REGION Network 2: TESTE CHACHA 20 ROUNDS
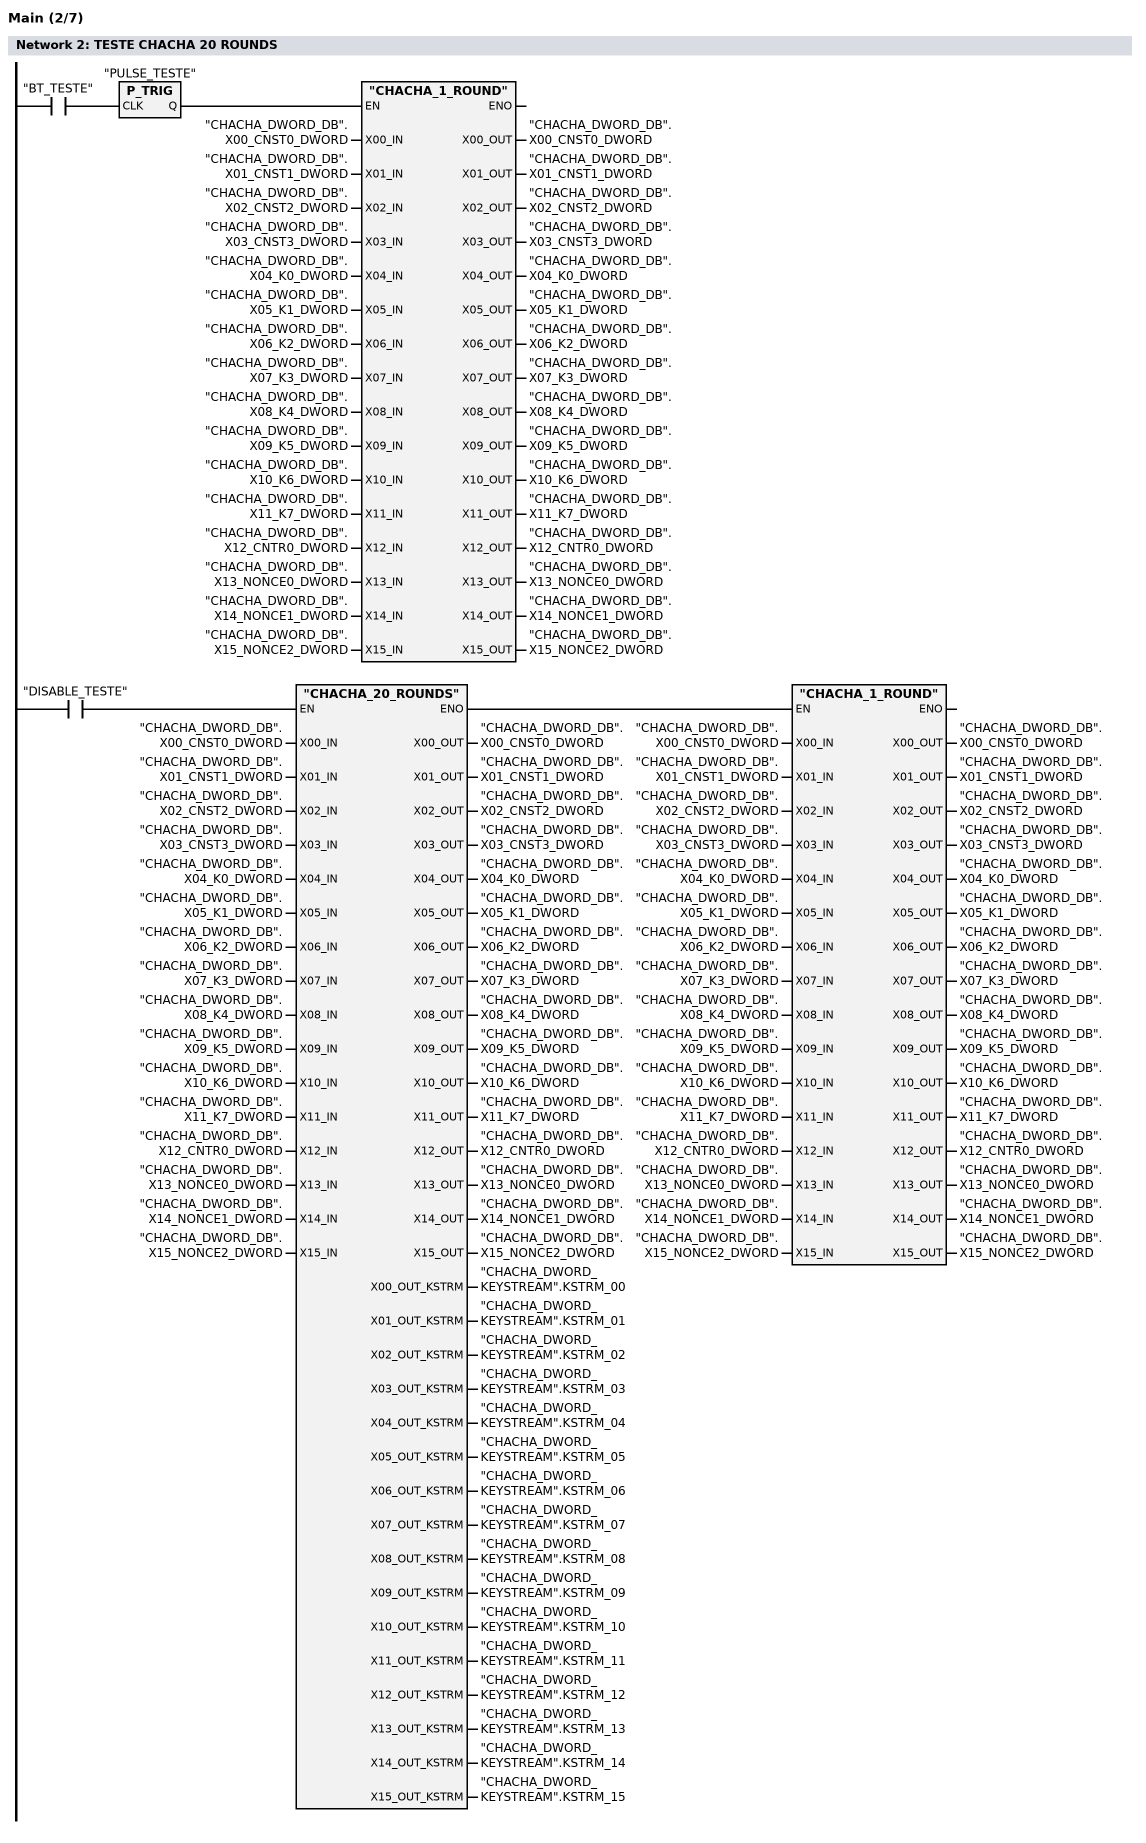
   RUNG wire#powerrail
      Contact( "BT_TESTE" )
      P_Trig( "PULSE_TESTE" )
      "CHACHA_1_ROUND"(X00_IN := "CHACHA_DWORD_DB".X00_CNST0_DWORD, X01_IN := "CHACHA_DWORD_DB".X01_CNST1_DWORD, X02_IN := "CHACHA_DWORD_DB".X02_CNST2_DWORD, X03_IN := "CHACHA_DWORD_DB".X03_CNST3_DWORD, X04_IN := "CHACHA_DWORD_DB".X04_K0_DWORD, X05_IN := "CHACHA_DWORD_DB".X05_K1_DWORD, X06_IN := "CHACHA_DWORD_DB".X06_K2_DWORD, X07_IN := "CHACHA_DWORD_DB".X07_K3_DWORD, X08_IN := "CHACHA_DWORD_DB".X08_K4_DWORD, X09_IN := "CHACHA_DWORD_DB".X09_K5_DWORD, X10_IN := "CHACHA_DWORD_DB".X10_K6_DWORD, X11_IN := "CHACHA_DWORD_DB".X11_K7_DWORD, X12_IN := "CHACHA_DWORD_DB".X12_CNTR0_DWORD, X13_IN := "CHACHA_DWORD_DB".X13_NONCE0_DWORD, X14_IN := "CHACHA_DWORD_DB".X14_NONCE1_DWORD, X15_IN := "CHACHA_DWORD_DB".X15_NONCE2_DWORD, X00_OUT => "CHACHA_DWORD_DB".X00_CNST0_DWORD, X01_OUT => "CHACHA_DWORD_DB".X01_CNST1_DWORD, X02_OUT => "CHACHA_DWORD_DB".X02_CNST2_DWORD, X03_OUT => "CHACHA_DWORD_DB".X03_CNST3_DWORD, X04_OUT => "CHACHA_DWORD_DB".X04_K0_DWORD, X05_OUT => "CHACHA_DWORD_DB".X05_K1_DWORD, X06_OUT => "CHACHA_DWORD_DB".X06_K2_DWORD, X07_OUT => "CHACHA_DWORD_DB".X07_K3_DWORD, X08_OUT => "CHACHA_DWORD_DB".X08_K4_DWORD, X09_OUT => "CHACHA_DWORD_DB".X09_K5_DWORD, X10_OUT => "CHACHA_DWORD_DB".X10_K6_DWORD, X11_OUT => "CHACHA_DWORD_DB".X11_K7_DWORD, X12_OUT => "CHACHA_DWORD_DB".X12_CNTR0_DWORD, X13_OUT => "CHACHA_DWORD_DB".X13_NONCE0_DWORD, X14_OUT => "CHACHA_DWORD_DB".X14_NONCE1_DWORD, X15_OUT => "CHACHA_DWORD_DB".X15_NONCE2_DWORD)
   END_RUNG
   RUNG wire#powerrail
      Contact( "DISABLE_TESTE" )
      "CHACHA_20_ROUNDS"(X00_IN := "CHACHA_DWORD_DB".X00_CNST0_DWORD, X01_IN := "CHACHA_DWORD_DB".X01_CNST1_DWORD, X02_IN := "CHACHA_DWORD_DB".X02_CNST2_DWORD, X03_IN := "CHACHA_DWORD_DB".X03_CNST3_DWORD, X04_IN := "CHACHA_DWORD_DB".X04_K0_DWORD, X05_IN := "CHACHA_DWORD_DB".X05_K1_DWORD, X06_IN := "CHACHA_DWORD_DB".X06_K2_DWORD, X07_IN := "CHACHA_DWORD_DB".X07_K3_DWORD, X08_IN := "CHACHA_DWORD_DB".X08_K4_DWORD, X09_IN := "CHACHA_DWORD_DB".X09_K5_DWORD, X10_IN := "CHACHA_DWORD_DB".X10_K6_DWORD, X11_IN := "CHACHA_DWORD_DB".X11_K7_DWORD, X12_IN := "CHACHA_DWORD_DB".X12_CNTR0_DWORD, X13_IN := "CHACHA_DWORD_DB".X13_NONCE0_DWORD, X14_IN := "CHACHA_DWORD_DB".X14_NONCE1_DWORD, X15_IN := "CHACHA_DWORD_DB".X15_NONCE2_DWORD, X00_OUT => "CHACHA_DWORD_DB".X00_CNST0_DWORD, X01_OUT => "CHACHA_DWORD_DB".X01_CNST1_DWORD, X02_OUT => "CHACHA_DWORD_DB".X02_CNST2_DWORD, X03_OUT => "CHACHA_DWORD_DB".X03_CNST3_DWORD, X04_OUT => "CHACHA_DWORD_DB".X04_K0_DWORD, X05_OUT => "CHACHA_DWORD_DB".X05_K1_DWORD, X06_OUT => "CHACHA_DWORD_DB".X06_K2_DWORD, X07_OUT => "CHACHA_DWORD_DB".X07_K3_DWORD, X08_OUT => "CHACHA_DWORD_DB".X08_K4_DWORD, X09_OUT => "CHACHA_DWORD_DB".X09_K5_DWORD, X10_OUT => "CHACHA_DWORD_DB".X10_K6_DWORD, X11_OUT => "CHACHA_DWORD_DB".X11_K7_DWORD, X12_OUT => "CHACHA_DWORD_DB".X12_CNTR0_DWORD, X13_OUT => "CHACHA_DWORD_DB".X13_NONCE0_DWORD, X14_OUT => "CHACHA_DWORD_DB".X14_NONCE1_DWORD, X15_OUT => "CHACHA_DWORD_DB".X15_NONCE2_DWORD, X00_OUT_KSTRM => "CHACHA_DWORD_KEYSTREAM".KSTRM_00, X01_OUT_KSTRM => "CHACHA_DWORD_KEYSTREAM".KSTRM_01, X02_OUT_KSTRM => "CHACHA_DWORD_KEYSTREAM".KSTRM_02, X03_OUT_KSTRM => "CHACHA_DWORD_KEYSTREAM".KSTRM_03, X04_OUT_KSTRM => "CHACHA_DWORD_KEYSTREAM".KSTRM_04, X05_OUT_KSTRM => "CHACHA_DWORD_KEYSTREAM".KSTRM_05, X06_OUT_KSTRM => "CHACHA_DWORD_KEYSTREAM".KSTRM_06, X07_OUT_KSTRM => "CHACHA_DWORD_KEYSTREAM".KSTRM_07, X08_OUT_KSTRM => "CHACHA_DWORD_KEYSTREAM".KSTRM_08, X09_OUT_KSTRM => "CHACHA_DWORD_KEYSTREAM".KSTRM_09, X10_OUT_KSTRM => "CHACHA_DWORD_KEYSTREAM".KSTRM_10, X11_OUT_KSTRM => "CHACHA_DWORD_KEYSTREAM".KSTRM_11, X12_OUT_KSTRM => "CHACHA_DWORD_KEYSTREAM".KSTRM_12, X13_OUT_KSTRM => "CHACHA_DWORD_KEYSTREAM".KSTRM_13, X14_OUT_KSTRM => "CHACHA_DWORD_KEYSTREAM".KSTRM_14, X15_OUT_KSTRM => "CHACHA_DWORD_KEYSTREAM".KSTRM_15)
      "CHACHA_1_ROUND"(X00_IN := "CHACHA_DWORD_DB".X00_CNST0_DWORD, X01_IN := "CHACHA_DWORD_DB".X01_CNST1_DWORD, X02_IN := "CHACHA_DWORD_DB".X02_CNST2_DWORD, X03_IN := "CHACHA_DWORD_DB".X03_CNST3_DWORD, X04_IN := "CHACHA_DWORD_DB".X04_K0_DWORD, X05_IN := "CHACHA_DWORD_DB".X05_K1_DWORD, X06_IN := "CHACHA_DWORD_DB".X06_K2_DWORD, X07_IN := "CHACHA_DWORD_DB".X07_K3_DWORD, X08_IN := "CHACHA_DWORD_DB".X08_K4_DWORD, X09_IN := "CHACHA_DWORD_DB".X09_K5_DWORD, X10_IN := "CHACHA_DWORD_DB".X10_K6_DWORD, X11_IN := "CHACHA_DWORD_DB".X11_K7_DWORD, X12_IN := "CHACHA_DWORD_DB".X12_CNTR0_DWORD, X13_IN := "CHACHA_DWORD_DB".X13_NONCE0_DWORD, X14_IN := "CHACHA_DWORD_DB".X14_NONCE1_DWORD, X15_IN := "CHACHA_DWORD_DB".X15_NONCE2_DWORD, X00_OUT => "CHACHA_DWORD_DB".X00_CNST0_DWORD, X01_OUT => "CHACHA_DWORD_DB".X01_CNST1_DWORD, X02_OUT => "CHACHA_DWORD_DB".X02_CNST2_DWORD, X03_OUT => "CHACHA_DWORD_DB".X03_CNST3_DWORD, X04_OUT => "CHACHA_DWORD_DB".X04_K0_DWORD, X05_OUT => "CHACHA_DWORD_DB".X05_K1_DWORD, X06_OUT => "CHACHA_DWORD_DB".X06_K2_DWORD, X07_OUT => "CHACHA_DWORD_DB".X07_K3_DWORD, X08_OUT => "CHACHA_DWORD_DB".X08_K4_DWORD, X09_OUT => "CHACHA_DWORD_DB".X09_K5_DWORD, X10_OUT => "CHACHA_DWORD_DB".X10_K6_DWORD, X11_OUT => "CHACHA_DWORD_DB".X11_K7_DWORD, X12_OUT => "CHACHA_DWORD_DB".X12_CNTR0_DWORD, X13_OUT => "CHACHA_DWORD_DB".X13_NONCE0_DWORD, X14_OUT => "CHACHA_DWORD_DB".X14_NONCE1_DWORD, X15_OUT => "CHACHA_DWORD_DB".X15_NONCE2_DWORD)
   END_RUNG
   // the same network as SCL:
   #_w1 := "BT_TESTE" AND NOT "PULSE_TESTE";   // rising edge
   "PULSE_TESTE" := "BT_TESTE";
   IF #_w1 THEN
       "CHACHA_1_ROUND"(X00_IN := "CHACHA_DWORD_DB".X00_CNST0_DWORD,
                        X01_IN := "CHACHA_DWORD_DB".X01_CNST1_DWORD,
                        X02_IN := "CHACHA_DWORD_DB".X02_CNST2_DWORD,
                        X03_IN := "CHACHA_DWORD_DB".X03_CNST3_DWORD,
                        X04_IN := "CHACHA_DWORD_DB".X04_K0_DWORD,
                        X05_IN := "CHACHA_DWORD_DB".X05_K1_DWORD,
                        X06_IN := "CHACHA_DWORD_DB".X06_K2_DWORD,
                        X07_IN := "CHACHA_DWORD_DB".X07_K3_DWORD,
                        X08_IN := "CHACHA_DWORD_DB".X08_K4_DWORD,
                        X09_IN := "CHACHA_DWORD_DB".X09_K5_DWORD,
                        X10_IN := "CHACHA_DWORD_DB".X10_K6_DWORD,
                        X11_IN := "CHACHA_DWORD_DB".X11_K7_DWORD,
                        X12_IN := "CHACHA_DWORD_DB".X12_CNTR0_DWORD,
                        X13_IN := "CHACHA_DWORD_DB".X13_NONCE0_DWORD,
                        X14_IN := "CHACHA_DWORD_DB".X14_NONCE1_DWORD,
                        X15_IN := "CHACHA_DWORD_DB".X15_NONCE2_DWORD,
                        X00_OUT => "CHACHA_DWORD_DB".X00_CNST0_DWORD,
                        X01_OUT => "CHACHA_DWORD_DB".X01_CNST1_DWORD,
                        X02_OUT => "CHACHA_DWORD_DB".X02_CNST2_DWORD,
                        X03_OUT => "CHACHA_DWORD_DB".X03_CNST3_DWORD,
                        X04_OUT => "CHACHA_DWORD_DB".X04_K0_DWORD,
                        X05_OUT => "CHACHA_DWORD_DB".X05_K1_DWORD,
                        X06_OUT => "CHACHA_DWORD_DB".X06_K2_DWORD,
                        X07_OUT => "CHACHA_DWORD_DB".X07_K3_DWORD,
                        X08_OUT => "CHACHA_DWORD_DB".X08_K4_DWORD,
                        X09_OUT => "CHACHA_DWORD_DB".X09_K5_DWORD,
                        X10_OUT => "CHACHA_DWORD_DB".X10_K6_DWORD,
                        X11_OUT => "CHACHA_DWORD_DB".X11_K7_DWORD,
                        X12_OUT => "CHACHA_DWORD_DB".X12_CNTR0_DWORD,
                        X13_OUT => "CHACHA_DWORD_DB".X13_NONCE0_DWORD,
                        X14_OUT => "CHACHA_DWORD_DB".X14_NONCE1_DWORD,
                        X15_OUT => "CHACHA_DWORD_DB".X15_NONCE2_DWORD);
   END_IF;
   "CHACHA_20_ROUNDS"(EN := "DISABLE_TESTE",
                      X00_IN := "CHACHA_DWORD_DB".X00_CNST0_DWORD,
                      X01_IN := "CHACHA_DWORD_DB".X01_CNST1_DWORD,
                      X02_IN := "CHACHA_DWORD_DB".X02_CNST2_DWORD,
                      X03_IN := "CHACHA_DWORD_DB".X03_CNST3_DWORD,
                      X04_IN := "CHACHA_DWORD_DB".X04_K0_DWORD,
                      X05_IN := "CHACHA_DWORD_DB".X05_K1_DWORD,
                      X06_IN := "CHACHA_DWORD_DB".X06_K2_DWORD,
                      X07_IN := "CHACHA_DWORD_DB".X07_K3_DWORD,
                      X08_IN := "CHACHA_DWORD_DB".X08_K4_DWORD,
                      X09_IN := "CHACHA_DWORD_DB".X09_K5_DWORD,
                      X10_IN := "CHACHA_DWORD_DB".X10_K6_DWORD,
                      X11_IN := "CHACHA_DWORD_DB".X11_K7_DWORD,
                      X12_IN := "CHACHA_DWORD_DB".X12_CNTR0_DWORD,
                      X13_IN := "CHACHA_DWORD_DB".X13_NONCE0_DWORD,
                      X14_IN := "CHACHA_DWORD_DB".X14_NONCE1_DWORD,
                      X15_IN := "CHACHA_DWORD_DB".X15_NONCE2_DWORD,
                      X00_OUT => "CHACHA_DWORD_DB".X00_CNST0_DWORD,
                      X01_OUT => "CHACHA_DWORD_DB".X01_CNST1_DWORD,
                      X02_OUT => "CHACHA_DWORD_DB".X02_CNST2_DWORD,
                      X03_OUT => "CHACHA_DWORD_DB".X03_CNST3_DWORD,
                      X04_OUT => "CHACHA_DWORD_DB".X04_K0_DWORD,
                      X05_OUT => "CHACHA_DWORD_DB".X05_K1_DWORD,
                      X06_OUT => "CHACHA_DWORD_DB".X06_K2_DWORD,
                      X07_OUT => "CHACHA_DWORD_DB".X07_K3_DWORD,
                      X08_OUT => "CHACHA_DWORD_DB".X08_K4_DWORD,
                      X09_OUT => "CHACHA_DWORD_DB".X09_K5_DWORD,
                      X10_OUT => "CHACHA_DWORD_DB".X10_K6_DWORD,
                      X11_OUT => "CHACHA_DWORD_DB".X11_K7_DWORD,
                      X12_OUT => "CHACHA_DWORD_DB".X12_CNTR0_DWORD,
                      X13_OUT => "CHACHA_DWORD_DB".X13_NONCE0_DWORD,
                      X14_OUT => "CHACHA_DWORD_DB".X14_NONCE1_DWORD,
                      X15_OUT => "CHACHA_DWORD_DB".X15_NONCE2_DWORD,
                      X00_OUT_KSTRM => "CHACHA_DWORD_KEYSTREAM".KSTRM_00,
                      X01_OUT_KSTRM => "CHACHA_DWORD_KEYSTREAM".KSTRM_01,
                      X02_OUT_KSTRM => "CHACHA_DWORD_KEYSTREAM".KSTRM_02,
                      X03_OUT_KSTRM => "CHACHA_DWORD_KEYSTREAM".KSTRM_03,
                      X04_OUT_KSTRM => "CHACHA_DWORD_KEYSTREAM".KSTRM_04,
                      X05_OUT_KSTRM => "CHACHA_DWORD_KEYSTREAM".KSTRM_05,
                      X06_OUT_KSTRM => "CHACHA_DWORD_KEYSTREAM".KSTRM_06,
                      X07_OUT_KSTRM => "CHACHA_DWORD_KEYSTREAM".KSTRM_07,
                      X08_OUT_KSTRM => "CHACHA_DWORD_KEYSTREAM".KSTRM_08,
                      X09_OUT_KSTRM => "CHACHA_DWORD_KEYSTREAM".KSTRM_09,
                      X10_OUT_KSTRM => "CHACHA_DWORD_KEYSTREAM".KSTRM_10,
                      X11_OUT_KSTRM => "CHACHA_DWORD_KEYSTREAM".KSTRM_11,
                      X12_OUT_KSTRM => "CHACHA_DWORD_KEYSTREAM".KSTRM_12,
                      X13_OUT_KSTRM => "CHACHA_DWORD_KEYSTREAM".KSTRM_13,
                      X14_OUT_KSTRM => "CHACHA_DWORD_KEYSTREAM".KSTRM_14,
                      X15_OUT_KSTRM => "CHACHA_DWORD_KEYSTREAM".KSTRM_15,
                      ENO => #_w2);
   IF #_w2 THEN
       "CHACHA_1_ROUND"(X00_IN := "CHACHA_DWORD_DB".X00_CNST0_DWORD,
                        X01_IN := "CHACHA_DWORD_DB".X01_CNST1_DWORD,
                        X02_IN := "CHACHA_DWORD_DB".X02_CNST2_DWORD,
                        X03_IN := "CHACHA_DWORD_DB".X03_CNST3_DWORD,
                        X04_IN := "CHACHA_DWORD_DB".X04_K0_DWORD,
                        X05_IN := "CHACHA_DWORD_DB".X05_K1_DWORD,
                        X06_IN := "CHACHA_DWORD_DB".X06_K2_DWORD,
                        X07_IN := "CHACHA_DWORD_DB".X07_K3_DWORD,
                        X08_IN := "CHACHA_DWORD_DB".X08_K4_DWORD,
                        X09_IN := "CHACHA_DWORD_DB".X09_K5_DWORD,
                        X10_IN := "CHACHA_DWORD_DB".X10_K6_DWORD,
                        X11_IN := "CHACHA_DWORD_DB".X11_K7_DWORD,
                        X12_IN := "CHACHA_DWORD_DB".X12_CNTR0_DWORD,
                        X13_IN := "CHACHA_DWORD_DB".X13_NONCE0_DWORD,
                        X14_IN := "CHACHA_DWORD_DB".X14_NONCE1_DWORD,
                        X15_IN := "CHACHA_DWORD_DB".X15_NONCE2_DWORD,
                        X00_OUT => "CHACHA_DWORD_DB".X00_CNST0_DWORD,
                        X01_OUT => "CHACHA_DWORD_DB".X01_CNST1_DWORD,
                        X02_OUT => "CHACHA_DWORD_DB".X02_CNST2_DWORD,
                        X03_OUT => "CHACHA_DWORD_DB".X03_CNST3_DWORD,
                        X04_OUT => "CHACHA_DWORD_DB".X04_K0_DWORD,
                        X05_OUT => "CHACHA_DWORD_DB".X05_K1_DWORD,
                        X06_OUT => "CHACHA_DWORD_DB".X06_K2_DWORD,
                        X07_OUT => "CHACHA_DWORD_DB".X07_K3_DWORD,
                        X08_OUT => "CHACHA_DWORD_DB".X08_K4_DWORD,
                        X09_OUT => "CHACHA_DWORD_DB".X09_K5_DWORD,
                        X10_OUT => "CHACHA_DWORD_DB".X10_K6_DWORD,
                        X11_OUT => "CHACHA_DWORD_DB".X11_K7_DWORD,
                        X12_OUT => "CHACHA_DWORD_DB".X12_CNTR0_DWORD,
                        X13_OUT => "CHACHA_DWORD_DB".X13_NONCE0_DWORD,
                        X14_OUT => "CHACHA_DWORD_DB".X14_NONCE1_DWORD,
                        X15_OUT => "CHACHA_DWORD_DB".X15_NONCE2_DWORD);
   END_IF;
END_REGION

REGION Network 3: TESTE CHACHA 20 ROUNDS - RUNTIME STOP
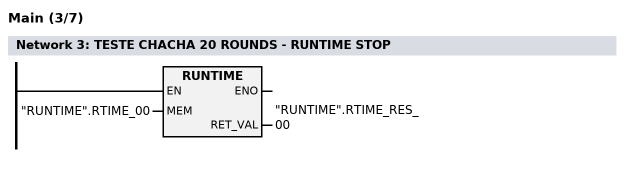
   // no SCL statement known for Runtime: written as a call
   "RUNTIME".RTIME_RES_00 := Runtime(mem := "RUNTIME".RTIME_00);
END_REGION

REGION Network 4: CHACHA QUANDO HABILITADO POR: TAG-TEMP-"ENABLE_CHACHA"
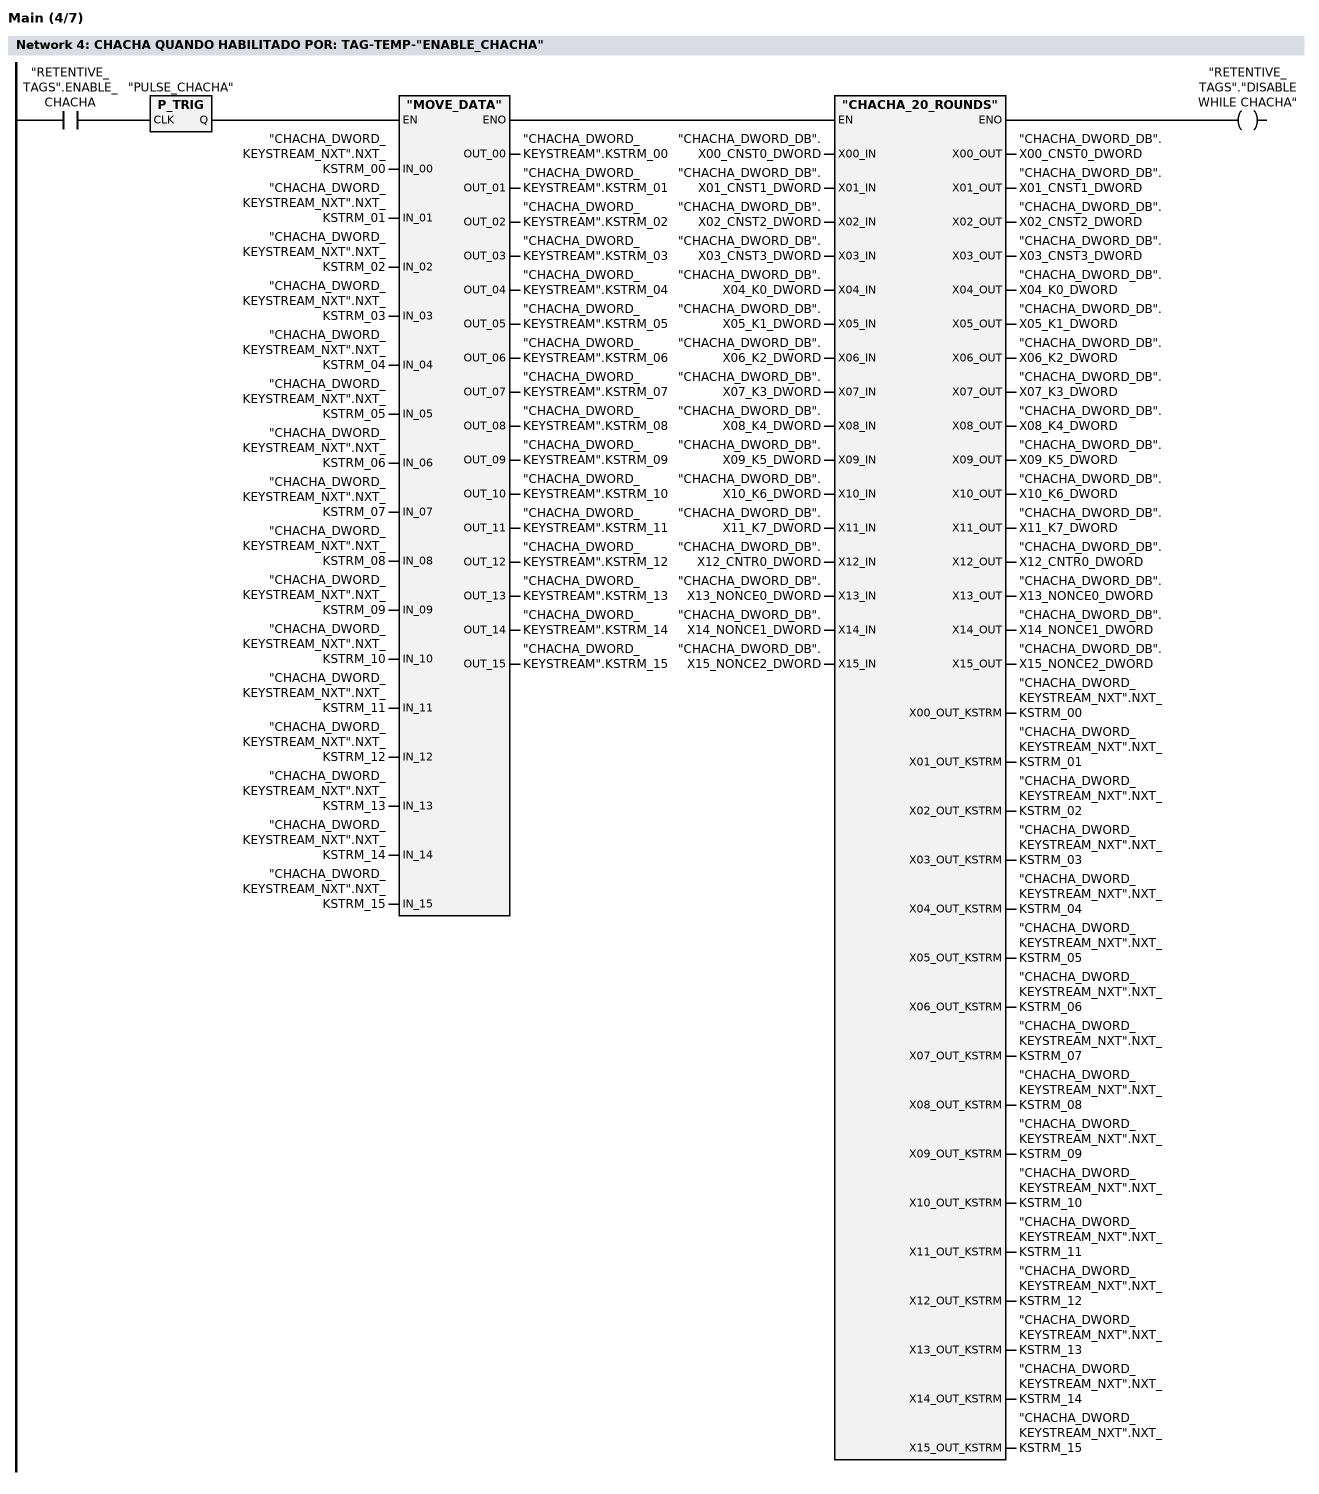
   RUNG wire#powerrail
      Contact( "RETENTIVE_TAGS".ENABLE_CHACHA )
      P_Trig( "PULSE_CHACHA" )
      "MOVE_DATA"(IN_00 := "CHACHA_DWORD_KEYSTREAM_NXT".NXT_KSTRM_00, IN_01 := "CHACHA_DWORD_KEYSTREAM_NXT".NXT_KSTRM_01, IN_02 := "CHACHA_DWORD_KEYSTREAM_NXT".NXT_KSTRM_02, IN_03 := "CHACHA_DWORD_KEYSTREAM_NXT".NXT_KSTRM_03, IN_04 := "CHACHA_DWORD_KEYSTREAM_NXT".NXT_KSTRM_04, IN_05 := "CHACHA_DWORD_KEYSTREAM_NXT".NXT_KSTRM_05, IN_06 := "CHACHA_DWORD_KEYSTREAM_NXT".NXT_KSTRM_06, IN_07 := "CHACHA_DWORD_KEYSTREAM_NXT".NXT_KSTRM_07, IN_08 := "CHACHA_DWORD_KEYSTREAM_NXT".NXT_KSTRM_08, IN_09 := "CHACHA_DWORD_KEYSTREAM_NXT".NXT_KSTRM_09, IN_10 := "CHACHA_DWORD_KEYSTREAM_NXT".NXT_KSTRM_10, IN_11 := "CHACHA_DWORD_KEYSTREAM_NXT".NXT_KSTRM_11, IN_12 := "CHACHA_DWORD_KEYSTREAM_NXT".NXT_KSTRM_12, IN_13 := "CHACHA_DWORD_KEYSTREAM_NXT".NXT_KSTRM_13, IN_14 := "CHACHA_DWORD_KEYSTREAM_NXT".NXT_KSTRM_14, IN_15 := "CHACHA_DWORD_KEYSTREAM_NXT".NXT_KSTRM_15, OUT_00 => "CHACHA_DWORD_KEYSTREAM".KSTRM_00, OUT_01 => "CHACHA_DWORD_KEYSTREAM".KSTRM_01, OUT_02 => "CHACHA_DWORD_KEYSTREAM".KSTRM_02, OUT_03 => "CHACHA_DWORD_KEYSTREAM".KSTRM_03, OUT_04 => "CHACHA_DWORD_KEYSTREAM".KSTRM_04, OUT_05 => "CHACHA_DWORD_KEYSTREAM".KSTRM_05, OUT_06 => "CHACHA_DWORD_KEYSTREAM".KSTRM_06, OUT_07 => "CHACHA_DWORD_KEYSTREAM".KSTRM_07, OUT_08 => "CHACHA_DWORD_KEYSTREAM".KSTRM_08, OUT_09 => "CHACHA_DWORD_KEYSTREAM".KSTRM_09, OUT_10 => "CHACHA_DWORD_KEYSTREAM".KSTRM_10, OUT_11 => "CHACHA_DWORD_KEYSTREAM".KSTRM_11, OUT_12 => "CHACHA_DWORD_KEYSTREAM".KSTRM_12, OUT_13 => "CHACHA_DWORD_KEYSTREAM".KSTRM_13, OUT_14 => "CHACHA_DWORD_KEYSTREAM".KSTRM_14, OUT_15 => "CHACHA_DWORD_KEYSTREAM".KSTRM_15)
      "CHACHA_20_ROUNDS"(X00_IN := "CHACHA_DWORD_DB".X00_CNST0_DWORD, X01_IN := "CHACHA_DWORD_DB".X01_CNST1_DWORD, X02_IN := "CHACHA_DWORD_DB".X02_CNST2_DWORD, X03_IN := "CHACHA_DWORD_DB".X03_CNST3_DWORD, X04_IN := "CHACHA_DWORD_DB".X04_K0_DWORD, X05_IN := "CHACHA_DWORD_DB".X05_K1_DWORD, X06_IN := "CHACHA_DWORD_DB".X06_K2_DWORD, X07_IN := "CHACHA_DWORD_DB".X07_K3_DWORD, X08_IN := "CHACHA_DWORD_DB".X08_K4_DWORD, X09_IN := "CHACHA_DWORD_DB".X09_K5_DWORD, X10_IN := "CHACHA_DWORD_DB".X10_K6_DWORD, X11_IN := "CHACHA_DWORD_DB".X11_K7_DWORD, X12_IN := "CHACHA_DWORD_DB".X12_CNTR0_DWORD, X13_IN := "CHACHA_DWORD_DB".X13_NONCE0_DWORD, X14_IN := "CHACHA_DWORD_DB".X14_NONCE1_DWORD, X15_IN := "CHACHA_DWORD_DB".X15_NONCE2_DWORD, X00_OUT => "CHACHA_DWORD_DB".X00_CNST0_DWORD, X01_OUT => "CHACHA_DWORD_DB".X01_CNST1_DWORD, X02_OUT => "CHACHA_DWORD_DB".X02_CNST2_DWORD, X03_OUT => "CHACHA_DWORD_DB".X03_CNST3_DWORD, X04_OUT => "CHACHA_DWORD_DB".X04_K0_DWORD, X05_OUT => "CHACHA_DWORD_DB".X05_K1_DWORD, X06_OUT => "CHACHA_DWORD_DB".X06_K2_DWORD, X07_OUT => "CHACHA_DWORD_DB".X07_K3_DWORD, X08_OUT => "CHACHA_DWORD_DB".X08_K4_DWORD, X09_OUT => "CHACHA_DWORD_DB".X09_K5_DWORD, X10_OUT => "CHACHA_DWORD_DB".X10_K6_DWORD, X11_OUT => "CHACHA_DWORD_DB".X11_K7_DWORD, X12_OUT => "CHACHA_DWORD_DB".X12_CNTR0_DWORD, X13_OUT => "CHACHA_DWORD_DB".X13_NONCE0_DWORD, X14_OUT => "CHACHA_DWORD_DB".X14_NONCE1_DWORD, X15_OUT => "CHACHA_DWORD_DB".X15_NONCE2_DWORD, X00_OUT_KSTRM => "CHACHA_DWORD_KEYSTREAM_NXT".NXT_KSTRM_00, X01_OUT_KSTRM => "CHACHA_DWORD_KEYSTREAM_NXT".NXT_KSTRM_01, X02_OUT_KSTRM => "CHACHA_DWORD_KEYSTREAM_NXT".NXT_KSTRM_02, X03_OUT_KSTRM => "CHACHA_DWORD_KEYSTREAM_NXT".NXT_KSTRM_03, X04_OUT_KSTRM => "CHACHA_DWORD_KEYSTREAM_NXT".NXT_KSTRM_04, X05_OUT_KSTRM => "CHACHA_DWORD_KEYSTREAM_NXT".NXT_KSTRM_05, X06_OUT_KSTRM => "CHACHA_DWORD_KEYSTREAM_NXT".NXT_KSTRM_06, X07_OUT_KSTRM => "CHACHA_DWORD_KEYSTREAM_NXT".NXT_KSTRM_07, X08_OUT_KSTRM => "CHACHA_DWORD_KEYSTREAM_NXT".NXT_KSTRM_08, X09_OUT_KSTRM => "CHACHA_DWORD_KEYSTREAM_NXT".NXT_KSTRM_09, X10_OUT_KSTRM => "CHACHA_DWORD_KEYSTREAM_NXT".NXT_KSTRM_10, X11_OUT_KSTRM => "CHACHA_DWORD_KEYSTREAM_NXT".NXT_KSTRM_11, X12_OUT_KSTRM => "CHACHA_DWORD_KEYSTREAM_NXT".NXT_KSTRM_12, X13_OUT_KSTRM => "CHACHA_DWORD_KEYSTREAM_NXT".NXT_KSTRM_13, X14_OUT_KSTRM => "CHACHA_DWORD_KEYSTREAM_NXT".NXT_KSTRM_14, X15_OUT_KSTRM => "CHACHA_DWORD_KEYSTREAM_NXT".NXT_KSTRM_15)
      Coil( "RETENTIVE_TAGS"."DISABLE WHILE CHACHA" )
   END_RUNG
   // the same network as SCL:
   #_w1 := "RETENTIVE_TAGS".ENABLE_CHACHA AND NOT "PULSE_CHACHA";   // rising edge
   "PULSE_CHACHA" := "RETENTIVE_TAGS".ENABLE_CHACHA;
   "MOVE_DATA"(EN := #_w1,
               IN_00 := "CHACHA_DWORD_KEYSTREAM_NXT".NXT_KSTRM_00,
               IN_01 := "CHACHA_DWORD_KEYSTREAM_NXT".NXT_KSTRM_01,
               IN_02 := "CHACHA_DWORD_KEYSTREAM_NXT".NXT_KSTRM_02,
               IN_03 := "CHACHA_DWORD_KEYSTREAM_NXT".NXT_KSTRM_03,
               IN_04 := "CHACHA_DWORD_KEYSTREAM_NXT".NXT_KSTRM_04,
               IN_05 := "CHACHA_DWORD_KEYSTREAM_NXT".NXT_KSTRM_05,
               IN_06 := "CHACHA_DWORD_KEYSTREAM_NXT".NXT_KSTRM_06,
               IN_07 := "CHACHA_DWORD_KEYSTREAM_NXT".NXT_KSTRM_07,
               IN_08 := "CHACHA_DWORD_KEYSTREAM_NXT".NXT_KSTRM_08,
               IN_09 := "CHACHA_DWORD_KEYSTREAM_NXT".NXT_KSTRM_09,
               IN_10 := "CHACHA_DWORD_KEYSTREAM_NXT".NXT_KSTRM_10,
               IN_11 := "CHACHA_DWORD_KEYSTREAM_NXT".NXT_KSTRM_11,
               IN_12 := "CHACHA_DWORD_KEYSTREAM_NXT".NXT_KSTRM_12,
               IN_13 := "CHACHA_DWORD_KEYSTREAM_NXT".NXT_KSTRM_13,
               IN_14 := "CHACHA_DWORD_KEYSTREAM_NXT".NXT_KSTRM_14,
               IN_15 := "CHACHA_DWORD_KEYSTREAM_NXT".NXT_KSTRM_15,
               OUT_00 => "CHACHA_DWORD_KEYSTREAM".KSTRM_00,
               OUT_01 => "CHACHA_DWORD_KEYSTREAM".KSTRM_01,
               OUT_02 => "CHACHA_DWORD_KEYSTREAM".KSTRM_02,
               OUT_03 => "CHACHA_DWORD_KEYSTREAM".KSTRM_03,
               OUT_04 => "CHACHA_DWORD_KEYSTREAM".KSTRM_04,
               OUT_05 => "CHACHA_DWORD_KEYSTREAM".KSTRM_05,
               OUT_06 => "CHACHA_DWORD_KEYSTREAM".KSTRM_06,
               OUT_07 => "CHACHA_DWORD_KEYSTREAM".KSTRM_07,
               OUT_08 => "CHACHA_DWORD_KEYSTREAM".KSTRM_08,
               OUT_09 => "CHACHA_DWORD_KEYSTREAM".KSTRM_09,
               OUT_10 => "CHACHA_DWORD_KEYSTREAM".KSTRM_10,
               OUT_11 => "CHACHA_DWORD_KEYSTREAM".KSTRM_11,
               OUT_12 => "CHACHA_DWORD_KEYSTREAM".KSTRM_12,
               OUT_13 => "CHACHA_DWORD_KEYSTREAM".KSTRM_13,
               OUT_14 => "CHACHA_DWORD_KEYSTREAM".KSTRM_14,
               OUT_15 => "CHACHA_DWORD_KEYSTREAM".KSTRM_15,
               ENO => #_w2);
   "CHACHA_20_ROUNDS"(EN := #_w2,
                      X00_IN := "CHACHA_DWORD_DB".X00_CNST0_DWORD,
                      X01_IN := "CHACHA_DWORD_DB".X01_CNST1_DWORD,
                      X02_IN := "CHACHA_DWORD_DB".X02_CNST2_DWORD,
                      X03_IN := "CHACHA_DWORD_DB".X03_CNST3_DWORD,
                      X04_IN := "CHACHA_DWORD_DB".X04_K0_DWORD,
                      X05_IN := "CHACHA_DWORD_DB".X05_K1_DWORD,
                      X06_IN := "CHACHA_DWORD_DB".X06_K2_DWORD,
                      X07_IN := "CHACHA_DWORD_DB".X07_K3_DWORD,
                      X08_IN := "CHACHA_DWORD_DB".X08_K4_DWORD,
                      X09_IN := "CHACHA_DWORD_DB".X09_K5_DWORD,
                      X10_IN := "CHACHA_DWORD_DB".X10_K6_DWORD,
                      X11_IN := "CHACHA_DWORD_DB".X11_K7_DWORD,
                      X12_IN := "CHACHA_DWORD_DB".X12_CNTR0_DWORD,
                      X13_IN := "CHACHA_DWORD_DB".X13_NONCE0_DWORD,
                      X14_IN := "CHACHA_DWORD_DB".X14_NONCE1_DWORD,
                      X15_IN := "CHACHA_DWORD_DB".X15_NONCE2_DWORD,
                      X00_OUT => "CHACHA_DWORD_DB".X00_CNST0_DWORD,
                      X01_OUT => "CHACHA_DWORD_DB".X01_CNST1_DWORD,
                      X02_OUT => "CHACHA_DWORD_DB".X02_CNST2_DWORD,
                      X03_OUT => "CHACHA_DWORD_DB".X03_CNST3_DWORD,
                      X04_OUT => "CHACHA_DWORD_DB".X04_K0_DWORD,
                      X05_OUT => "CHACHA_DWORD_DB".X05_K1_DWORD,
                      X06_OUT => "CHACHA_DWORD_DB".X06_K2_DWORD,
                      X07_OUT => "CHACHA_DWORD_DB".X07_K3_DWORD,
                      X08_OUT => "CHACHA_DWORD_DB".X08_K4_DWORD,
                      X09_OUT => "CHACHA_DWORD_DB".X09_K5_DWORD,
                      X10_OUT => "CHACHA_DWORD_DB".X10_K6_DWORD,
                      X11_OUT => "CHACHA_DWORD_DB".X11_K7_DWORD,
                      X12_OUT => "CHACHA_DWORD_DB".X12_CNTR0_DWORD,
                      X13_OUT => "CHACHA_DWORD_DB".X13_NONCE0_DWORD,
                      X14_OUT => "CHACHA_DWORD_DB".X14_NONCE1_DWORD,
                      X15_OUT => "CHACHA_DWORD_DB".X15_NONCE2_DWORD,
                      X00_OUT_KSTRM => "CHACHA_DWORD_KEYSTREAM_NXT".NXT_KSTRM_00,
                      X01_OUT_KSTRM => "CHACHA_DWORD_KEYSTREAM_NXT".NXT_KSTRM_01,
                      X02_OUT_KSTRM => "CHACHA_DWORD_KEYSTREAM_NXT".NXT_KSTRM_02,
                      X03_OUT_KSTRM => "CHACHA_DWORD_KEYSTREAM_NXT".NXT_KSTRM_03,
                      X04_OUT_KSTRM => "CHACHA_DWORD_KEYSTREAM_NXT".NXT_KSTRM_04,
                      X05_OUT_KSTRM => "CHACHA_DWORD_KEYSTREAM_NXT".NXT_KSTRM_05,
                      X06_OUT_KSTRM => "CHACHA_DWORD_KEYSTREAM_NXT".NXT_KSTRM_06,
                      X07_OUT_KSTRM => "CHACHA_DWORD_KEYSTREAM_NXT".NXT_KSTRM_07,
                      X08_OUT_KSTRM => "CHACHA_DWORD_KEYSTREAM_NXT".NXT_KSTRM_08,
                      X09_OUT_KSTRM => "CHACHA_DWORD_KEYSTREAM_NXT".NXT_KSTRM_09,
                      X10_OUT_KSTRM => "CHACHA_DWORD_KEYSTREAM_NXT".NXT_KSTRM_10,
                      X11_OUT_KSTRM => "CHACHA_DWORD_KEYSTREAM_NXT".NXT_KSTRM_11,
                      X12_OUT_KSTRM => "CHACHA_DWORD_KEYSTREAM_NXT".NXT_KSTRM_12,
                      X13_OUT_KSTRM => "CHACHA_DWORD_KEYSTREAM_NXT".NXT_KSTRM_13,
                      X14_OUT_KSTRM => "CHACHA_DWORD_KEYSTREAM_NXT".NXT_KSTRM_14,
                      X15_OUT_KSTRM => "CHACHA_DWORD_KEYSTREAM_NXT".NXT_KSTRM_15,
                      ENO => #_w3);
   "RETENTIVE_TAGS"."DISABLE WHILE CHACHA" := #_w3;
END_REGION

REGION Network 5: ATRIBUICOES DE VALORES NO PLAINTEXT
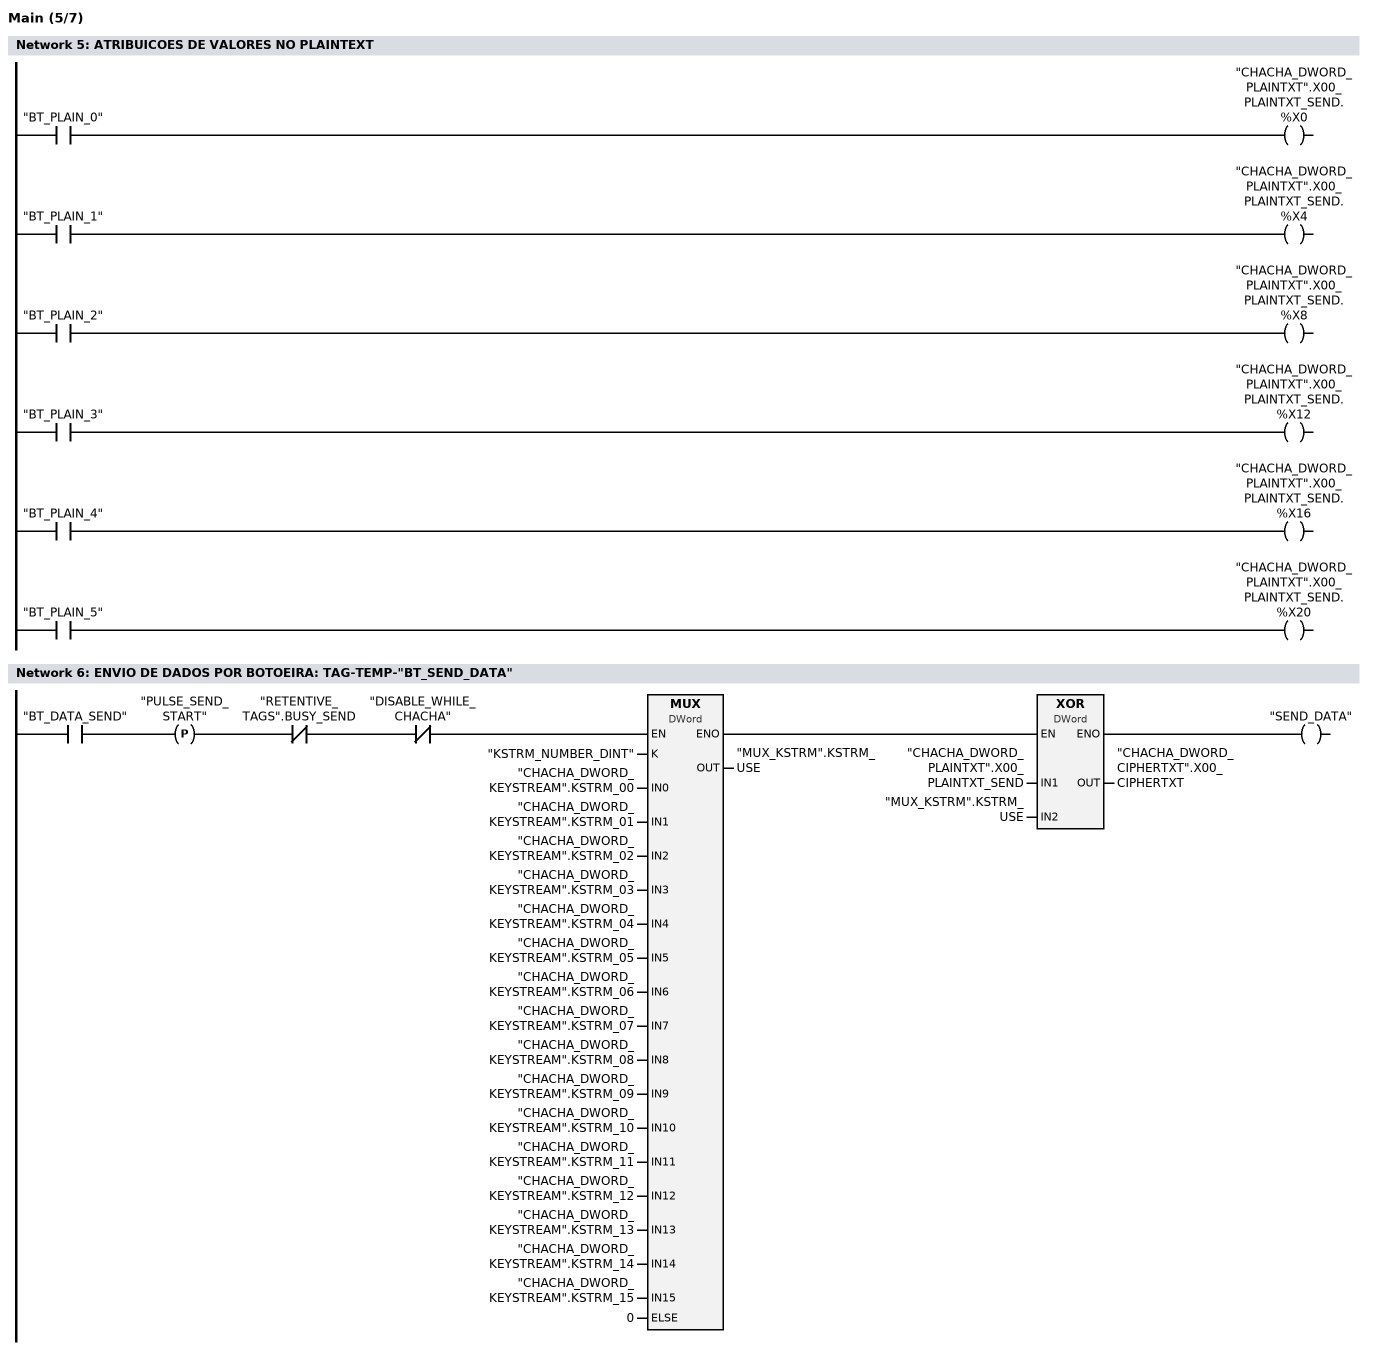
   RUNG wire#powerrail
      Contact( "BT_PLAIN_0" )
      Coil( "CHACHA_DWORD_PLAINTXT".X00_PLAINTXT_SEND.%X0 )
   END_RUNG
   RUNG wire#powerrail
      Contact( "BT_PLAIN_1" )
      Coil( "CHACHA_DWORD_PLAINTXT".X00_PLAINTXT_SEND.%X4 )
   END_RUNG
   RUNG wire#powerrail
      Contact( "BT_PLAIN_2" )
      Coil( "CHACHA_DWORD_PLAINTXT".X00_PLAINTXT_SEND.%X8 )
   END_RUNG
   RUNG wire#powerrail
      Contact( "BT_PLAIN_3" )
      Coil( "CHACHA_DWORD_PLAINTXT".X00_PLAINTXT_SEND.%X12 )
   END_RUNG
   RUNG wire#powerrail
      Contact( "BT_PLAIN_4" )
      Coil( "CHACHA_DWORD_PLAINTXT".X00_PLAINTXT_SEND.%X16 )
   END_RUNG
   RUNG wire#powerrail
      Contact( "BT_PLAIN_5" )
      Coil( "CHACHA_DWORD_PLAINTXT".X00_PLAINTXT_SEND.%X20 )
   END_RUNG
   // the same network as SCL:
   "CHACHA_DWORD_PLAINTXT".X00_PLAINTXT_SEND.%X0 := "BT_PLAIN_0";
   "CHACHA_DWORD_PLAINTXT".X00_PLAINTXT_SEND.%X4 := "BT_PLAIN_1";
   "CHACHA_DWORD_PLAINTXT".X00_PLAINTXT_SEND.%X8 := "BT_PLAIN_2";
   "CHACHA_DWORD_PLAINTXT".X00_PLAINTXT_SEND.%X12 := "BT_PLAIN_3";
   "CHACHA_DWORD_PLAINTXT".X00_PLAINTXT_SEND.%X16 := "BT_PLAIN_4";
   "CHACHA_DWORD_PLAINTXT".X00_PLAINTXT_SEND.%X20 := "BT_PLAIN_5";
END_REGION

REGION Network 6: ENVIO DE DADOS POR BOTOEIRA: TAG-TEMP-"BT_SEND_DATA"
   // no SCL statement known for Mux: written as a call
   // ENO of a box is taken as its EN; it also drops when the box reports an error
   #_w1 := "BT_DATA_SEND" AND NOT "PULSE_SEND_START";   // rising edge
   "PULSE_SEND_START" := "BT_DATA_SEND";
   #_w2 := #_w1 AND NOT "RETENTIVE_TAGS".BUSY_SEND AND NOT "DISABLE_WHILE_CHACHA";
   IF #_w2 THEN
       Mux(k := "KSTRM_NUMBER_DINT",
           in0 := "CHACHA_DWORD_KEYSTREAM".KSTRM_00,
           in1 := "CHACHA_DWORD_KEYSTREAM".KSTRM_01,
           in2 := "CHACHA_DWORD_KEYSTREAM".KSTRM_02,
           in3 := "CHACHA_DWORD_KEYSTREAM".KSTRM_03,
           in4 := "CHACHA_DWORD_KEYSTREAM".KSTRM_04,
           in5 := "CHACHA_DWORD_KEYSTREAM".KSTRM_05,
           in6 := "CHACHA_DWORD_KEYSTREAM".KSTRM_06,
           in7 := "CHACHA_DWORD_KEYSTREAM".KSTRM_07,
           in8 := "CHACHA_DWORD_KEYSTREAM".KSTRM_08,
           in9 := "CHACHA_DWORD_KEYSTREAM".KSTRM_09,
           in10 := "CHACHA_DWORD_KEYSTREAM".KSTRM_10,
           in11 := "CHACHA_DWORD_KEYSTREAM".KSTRM_11,
           in12 := "CHACHA_DWORD_KEYSTREAM".KSTRM_12,
           in13 := "CHACHA_DWORD_KEYSTREAM".KSTRM_13,
           in14 := "CHACHA_DWORD_KEYSTREAM".KSTRM_14,
           in15 := "CHACHA_DWORD_KEYSTREAM".KSTRM_15,
           "else" := 0,
           out => "MUX_KSTRM".KSTRM_USE);
       "CHACHA_DWORD_CIPHERTXT".X00_CIPHERTXT := "CHACHA_DWORD_PLAINTXT".X00_PLAINTXT_SEND XOR "MUX_KSTRM".KSTRM_USE;
   END_IF;
   "SEND_DATA" := #_w2;
END_REGION

REGION Network 7: BLOCO TSEND DE ENVIO DE DADOS
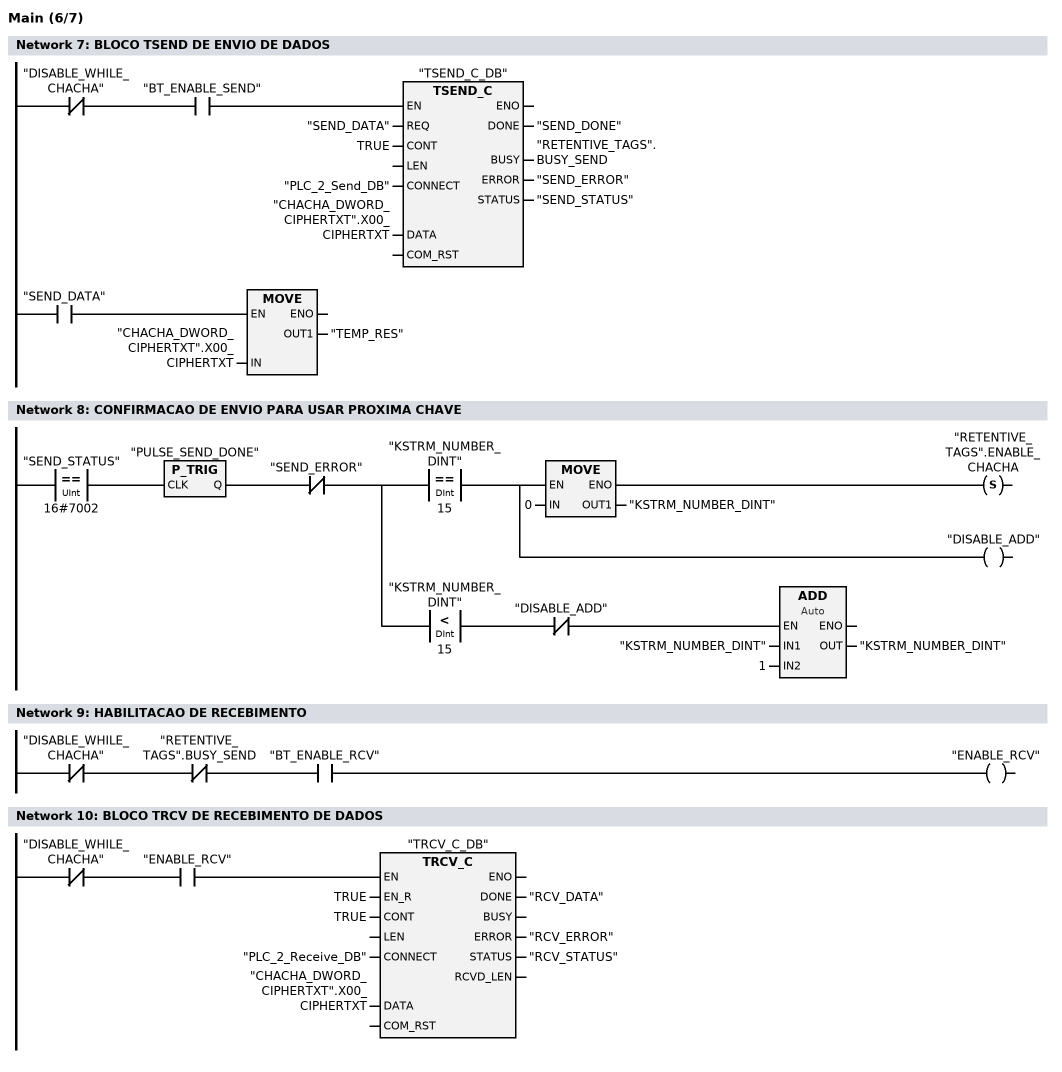
   IF NOT "DISABLE_WHILE_CHACHA" AND "BT_ENABLE_SEND" THEN
       "TSEND_C_DB"(REQ := "SEND_DATA",   // TSEND_C
                    CONT := TRUE,
                    CONNECT := "PLC_2_Send_DB",
                    DATA := "CHACHA_DWORD_CIPHERTXT".X00_CIPHERTXT,
                    DONE => "SEND_DONE",
                    BUSY => "RETENTIVE_TAGS".BUSY_SEND,
                    ERROR => "SEND_ERROR",
                    STATUS => "SEND_STATUS");
   END_IF;
   IF "SEND_DATA" THEN "TEMP_RES" := "CHACHA_DWORD_CIPHERTXT".X00_CIPHERTXT; END_IF;
END_REGION

REGION Network 8: CONFIRMACAO DE ENVIO PARA USAR PROXIMA CHAVE
   RUNG wire#powerrail
      { S7_Templates := "SrcType := UInt" } EQ_Contact(in1 := "SEND_STATUS", in2 := 16#7002)
      P_Trig( "PULSE_SEND_DONE" )
      I_Contact( "SEND_ERROR" )
      wire#w1
      { S7_Templates := "SrcType := DInt" } EQ_Contact(in1 := "KSTRM_NUMBER_DINT", in2 := 15)
      wire#w2
      { S7_GenerateENO := "TRUE" } Move(in := 0, out1 => "KSTRM_NUMBER_DINT")
      S_Coil( "RETENTIVE_TAGS".ENABLE_CHACHA )
   END_RUNG
   RUNG wire#w2
      Coil( "DISABLE_ADD" )
   END_RUNG
   RUNG wire#w1
      { S7_Templates := "SrcType := DInt" } LT_Contact(in1 := "KSTRM_NUMBER_DINT", in2 := 15)
      I_Contact( "DISABLE_ADD" )
      { S7_GenerateENO := "TRUE" } Add(in1 := "KSTRM_NUMBER_DINT", in2 := 1, out => "KSTRM_NUMBER_DINT")
   END_RUNG
   // the same network as SCL:
   // ENO of a box is taken as its EN; it also drops when the box reports an error
   #_w1 := "SEND_STATUS" = 16#7002;
   #_w2 := #_w1 AND NOT "PULSE_SEND_DONE";   // rising edge
   "PULSE_SEND_DONE" := #_w1;
   #_w3 := #_w2 AND NOT "SEND_ERROR";
   #_w4 := #_w3 AND ("KSTRM_NUMBER_DINT" = 15);
   IF #_w4 THEN
       "KSTRM_NUMBER_DINT" := 0;
       "RETENTIVE_TAGS".ENABLE_CHACHA := TRUE;
   END_IF;
   "DISABLE_ADD" := #_w4;
   IF #_w3 AND ("KSTRM_NUMBER_DINT" < 15) AND NOT "DISABLE_ADD" THEN
       "KSTRM_NUMBER_DINT" := "KSTRM_NUMBER_DINT" + 1;
   END_IF;
END_REGION

REGION Network 9: HABILITACAO DE RECEBIMENTO
   RUNG wire#powerrail
      I_Contact( "DISABLE_WHILE_CHACHA" )
      I_Contact( "RETENTIVE_TAGS".BUSY_SEND )
      Contact( "BT_ENABLE_RCV" )
      Coil( "ENABLE_RCV" )
   END_RUNG
   // the same network as SCL:
   "ENABLE_RCV" := NOT "DISABLE_WHILE_CHACHA" AND NOT "RETENTIVE_TAGS".BUSY_SEND AND "BT_ENABLE_RCV";
END_REGION

REGION Network 10: BLOCO TRCV DE RECEBIMENTO DE DADOS
   IF NOT "DISABLE_WHILE_CHACHA" AND "ENABLE_RCV" THEN
       "TRCV_C_DB"(EN_R := TRUE,   // TRCV_C
                   CONT := TRUE,
                   CONNECT := "PLC_2_Receive_DB",
                   DATA := "CHACHA_DWORD_CIPHERTXT".X00_CIPHERTXT,
                   DONE => "RCV_DATA",
                   ERROR => "RCV_ERROR",
                   STATUS => "RCV_STATUS");
   END_IF;
END_REGION

REGION Network 11: DECIFRAGEM DOS DADOS RECEBIDOS NO BLOCO TRCV
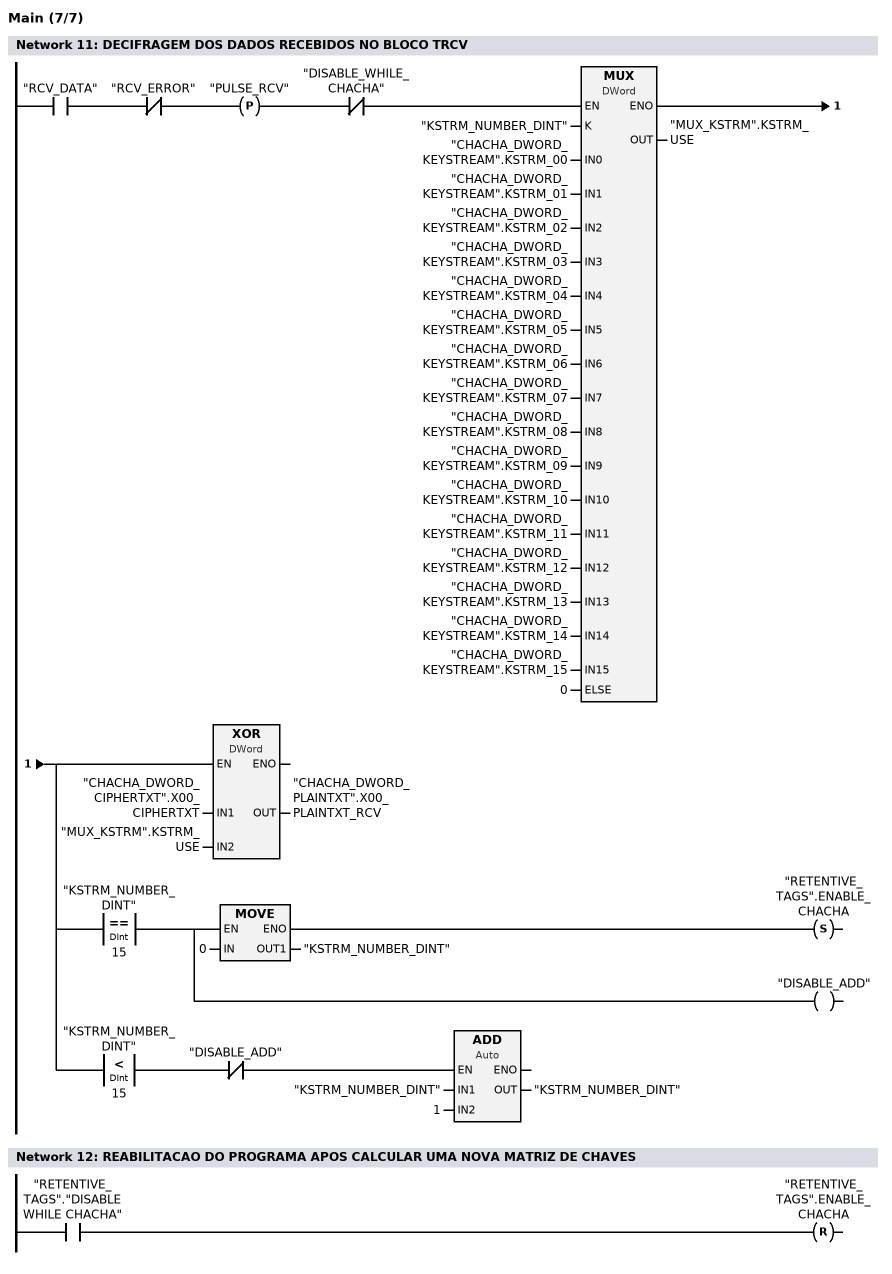
   // no SCL statement known for Mux: written as a call
   // ENO of a box is taken as its EN; it also drops when the box reports an error
   #_w1 := "RCV_DATA" AND NOT "RCV_ERROR";
   #_w2 := #_w1 AND NOT "PULSE_RCV";   // rising edge
   "PULSE_RCV" := #_w1;
   #_w3 := #_w2 AND NOT "DISABLE_WHILE_CHACHA";
   IF #_w3 THEN
       Mux(k := "KSTRM_NUMBER_DINT",
           in0 := "CHACHA_DWORD_KEYSTREAM".KSTRM_00,
           in1 := "CHACHA_DWORD_KEYSTREAM".KSTRM_01,
           in2 := "CHACHA_DWORD_KEYSTREAM".KSTRM_02,
           in3 := "CHACHA_DWORD_KEYSTREAM".KSTRM_03,
           in4 := "CHACHA_DWORD_KEYSTREAM".KSTRM_04,
           in5 := "CHACHA_DWORD_KEYSTREAM".KSTRM_05,
           in6 := "CHACHA_DWORD_KEYSTREAM".KSTRM_06,
           in7 := "CHACHA_DWORD_KEYSTREAM".KSTRM_07,
           in8 := "CHACHA_DWORD_KEYSTREAM".KSTRM_08,
           in9 := "CHACHA_DWORD_KEYSTREAM".KSTRM_09,
           in10 := "CHACHA_DWORD_KEYSTREAM".KSTRM_10,
           in11 := "CHACHA_DWORD_KEYSTREAM".KSTRM_11,
           in12 := "CHACHA_DWORD_KEYSTREAM".KSTRM_12,
           in13 := "CHACHA_DWORD_KEYSTREAM".KSTRM_13,
           in14 := "CHACHA_DWORD_KEYSTREAM".KSTRM_14,
           in15 := "CHACHA_DWORD_KEYSTREAM".KSTRM_15,
           "else" := 0,
           out => "MUX_KSTRM".KSTRM_USE);
       "CHACHA_DWORD_PLAINTXT".X00_PLAINTXT_RCV := "CHACHA_DWORD_CIPHERTXT".X00_CIPHERTXT XOR "MUX_KSTRM".KSTRM_USE;
   END_IF;
   #_w4 := #_w3 AND ("KSTRM_NUMBER_DINT" = 15);
   IF #_w4 THEN
       "KSTRM_NUMBER_DINT" := 0;
       "RETENTIVE_TAGS".ENABLE_CHACHA := TRUE;
   END_IF;
   "DISABLE_ADD" := #_w4;
   IF #_w3 AND ("KSTRM_NUMBER_DINT" < 15) AND NOT "DISABLE_ADD" THEN
       "KSTRM_NUMBER_DINT" := "KSTRM_NUMBER_DINT" + 1;
   END_IF;
END_REGION

REGION Network 12: REABILITACAO DO PROGRAMA APOS CALCULAR UMA NOVA MATRIZ DE CHAVES
   RUNG wire#powerrail
      Contact( "RETENTIVE_TAGS"."DISABLE WHILE CHACHA" )
      R_Coil( "RETENTIVE_TAGS".ENABLE_CHACHA )
   END_RUNG
   // the same network as SCL:
   IF "RETENTIVE_TAGS"."DISABLE WHILE CHACHA" THEN "RETENTIVE_TAGS".ENABLE_CHACHA := FALSE; END_IF;
END_REGION
END_ORGANIZATION_BLOCK

ORGANIZATION_BLOCK "Startup"   // OB100, LAD, Startup
TITLE = "Complete Restart"
{ S7_Optimized_Access := 'TRUE' }
VERSION : 0.1
   VAR_INPUT
      LostRetentive : Bool;   // True if retentive data are lost
      LostRTC : Bool;   // True if date and time are lost
   END_VAR
   VAR_TEMP   // added for the SCL form of the ladder/FBD networks
      _w1 : Bool;
   END_VAR
BEGIN

REGION Network 1
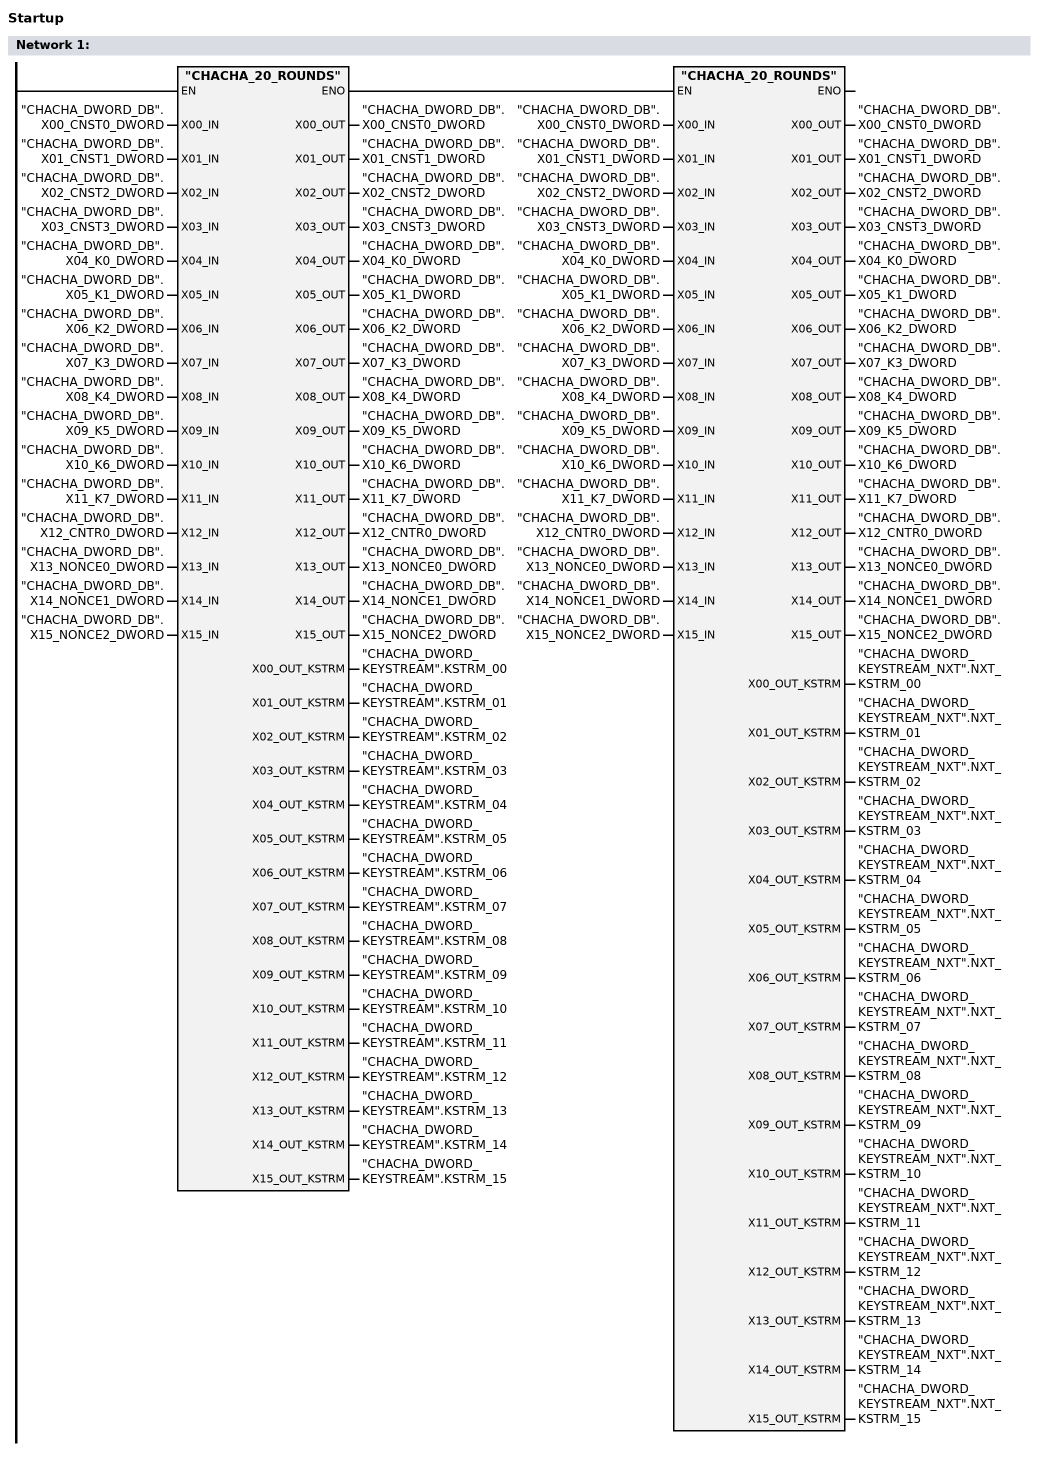
   RUNG wire#powerrail
      "CHACHA_20_ROUNDS"(X00_IN := "CHACHA_DWORD_DB".X00_CNST0_DWORD, X01_IN := "CHACHA_DWORD_DB".X01_CNST1_DWORD, X02_IN := "CHACHA_DWORD_DB".X02_CNST2_DWORD, X03_IN := "CHACHA_DWORD_DB".X03_CNST3_DWORD, X04_IN := "CHACHA_DWORD_DB".X04_K0_DWORD, X05_IN := "CHACHA_DWORD_DB".X05_K1_DWORD, X06_IN := "CHACHA_DWORD_DB".X06_K2_DWORD, X07_IN := "CHACHA_DWORD_DB".X07_K3_DWORD, X08_IN := "CHACHA_DWORD_DB".X08_K4_DWORD, X09_IN := "CHACHA_DWORD_DB".X09_K5_DWORD, X10_IN := "CHACHA_DWORD_DB".X10_K6_DWORD, X11_IN := "CHACHA_DWORD_DB".X11_K7_DWORD, X12_IN := "CHACHA_DWORD_DB".X12_CNTR0_DWORD, X13_IN := "CHACHA_DWORD_DB".X13_NONCE0_DWORD, X14_IN := "CHACHA_DWORD_DB".X14_NONCE1_DWORD, X15_IN := "CHACHA_DWORD_DB".X15_NONCE2_DWORD, X00_OUT => "CHACHA_DWORD_DB".X00_CNST0_DWORD, X01_OUT => "CHACHA_DWORD_DB".X01_CNST1_DWORD, X02_OUT => "CHACHA_DWORD_DB".X02_CNST2_DWORD, X03_OUT => "CHACHA_DWORD_DB".X03_CNST3_DWORD, X04_OUT => "CHACHA_DWORD_DB".X04_K0_DWORD, X05_OUT => "CHACHA_DWORD_DB".X05_K1_DWORD, X06_OUT => "CHACHA_DWORD_DB".X06_K2_DWORD, X07_OUT => "CHACHA_DWORD_DB".X07_K3_DWORD, X08_OUT => "CHACHA_DWORD_DB".X08_K4_DWORD, X09_OUT => "CHACHA_DWORD_DB".X09_K5_DWORD, X10_OUT => "CHACHA_DWORD_DB".X10_K6_DWORD, X11_OUT => "CHACHA_DWORD_DB".X11_K7_DWORD, X12_OUT => "CHACHA_DWORD_DB".X12_CNTR0_DWORD, X13_OUT => "CHACHA_DWORD_DB".X13_NONCE0_DWORD, X14_OUT => "CHACHA_DWORD_DB".X14_NONCE1_DWORD, X15_OUT => "CHACHA_DWORD_DB".X15_NONCE2_DWORD, X00_OUT_KSTRM => "CHACHA_DWORD_KEYSTREAM".KSTRM_00, X01_OUT_KSTRM => "CHACHA_DWORD_KEYSTREAM".KSTRM_01, X02_OUT_KSTRM => "CHACHA_DWORD_KEYSTREAM".KSTRM_02, X03_OUT_KSTRM => "CHACHA_DWORD_KEYSTREAM".KSTRM_03, X04_OUT_KSTRM => "CHACHA_DWORD_KEYSTREAM".KSTRM_04, X05_OUT_KSTRM => "CHACHA_DWORD_KEYSTREAM".KSTRM_05, X06_OUT_KSTRM => "CHACHA_DWORD_KEYSTREAM".KSTRM_06, X07_OUT_KSTRM => "CHACHA_DWORD_KEYSTREAM".KSTRM_07, X08_OUT_KSTRM => "CHACHA_DWORD_KEYSTREAM".KSTRM_08, X09_OUT_KSTRM => "CHACHA_DWORD_KEYSTREAM".KSTRM_09, X10_OUT_KSTRM => "CHACHA_DWORD_KEYSTREAM".KSTRM_10, X11_OUT_KSTRM => "CHACHA_DWORD_KEYSTREAM".KSTRM_11, X12_OUT_KSTRM => "CHACHA_DWORD_KEYSTREAM".KSTRM_12, X13_OUT_KSTRM => "CHACHA_DWORD_KEYSTREAM".KSTRM_13, X14_OUT_KSTRM => "CHACHA_DWORD_KEYSTREAM".KSTRM_14, X15_OUT_KSTRM => "CHACHA_DWORD_KEYSTREAM".KSTRM_15)
      "CHACHA_20_ROUNDS"(X00_IN := "CHACHA_DWORD_DB".X00_CNST0_DWORD, X01_IN := "CHACHA_DWORD_DB".X01_CNST1_DWORD, X02_IN := "CHACHA_DWORD_DB".X02_CNST2_DWORD, X03_IN := "CHACHA_DWORD_DB".X03_CNST3_DWORD, X04_IN := "CHACHA_DWORD_DB".X04_K0_DWORD, X05_IN := "CHACHA_DWORD_DB".X05_K1_DWORD, X06_IN := "CHACHA_DWORD_DB".X06_K2_DWORD, X07_IN := "CHACHA_DWORD_DB".X07_K3_DWORD, X08_IN := "CHACHA_DWORD_DB".X08_K4_DWORD, X09_IN := "CHACHA_DWORD_DB".X09_K5_DWORD, X10_IN := "CHACHA_DWORD_DB".X10_K6_DWORD, X11_IN := "CHACHA_DWORD_DB".X11_K7_DWORD, X12_IN := "CHACHA_DWORD_DB".X12_CNTR0_DWORD, X13_IN := "CHACHA_DWORD_DB".X13_NONCE0_DWORD, X14_IN := "CHACHA_DWORD_DB".X14_NONCE1_DWORD, X15_IN := "CHACHA_DWORD_DB".X15_NONCE2_DWORD, X00_OUT => "CHACHA_DWORD_DB".X00_CNST0_DWORD, X01_OUT => "CHACHA_DWORD_DB".X01_CNST1_DWORD, X02_OUT => "CHACHA_DWORD_DB".X02_CNST2_DWORD, X03_OUT => "CHACHA_DWORD_DB".X03_CNST3_DWORD, X04_OUT => "CHACHA_DWORD_DB".X04_K0_DWORD, X05_OUT => "CHACHA_DWORD_DB".X05_K1_DWORD, X06_OUT => "CHACHA_DWORD_DB".X06_K2_DWORD, X07_OUT => "CHACHA_DWORD_DB".X07_K3_DWORD, X08_OUT => "CHACHA_DWORD_DB".X08_K4_DWORD, X09_OUT => "CHACHA_DWORD_DB".X09_K5_DWORD, X10_OUT => "CHACHA_DWORD_DB".X10_K6_DWORD, X11_OUT => "CHACHA_DWORD_DB".X11_K7_DWORD, X12_OUT => "CHACHA_DWORD_DB".X12_CNTR0_DWORD, X13_OUT => "CHACHA_DWORD_DB".X13_NONCE0_DWORD, X14_OUT => "CHACHA_DWORD_DB".X14_NONCE1_DWORD, X15_OUT => "CHACHA_DWORD_DB".X15_NONCE2_DWORD, X00_OUT_KSTRM => "CHACHA_DWORD_KEYSTREAM_NXT".NXT_KSTRM_00, X01_OUT_KSTRM => "CHACHA_DWORD_KEYSTREAM_NXT".NXT_KSTRM_01, X02_OUT_KSTRM => "CHACHA_DWORD_KEYSTREAM_NXT".NXT_KSTRM_02, X03_OUT_KSTRM => "CHACHA_DWORD_KEYSTREAM_NXT".NXT_KSTRM_03, X04_OUT_KSTRM => "CHACHA_DWORD_KEYSTREAM_NXT".NXT_KSTRM_04, X05_OUT_KSTRM => "CHACHA_DWORD_KEYSTREAM_NXT".NXT_KSTRM_05, X06_OUT_KSTRM => "CHACHA_DWORD_KEYSTREAM_NXT".NXT_KSTRM_06, X07_OUT_KSTRM => "CHACHA_DWORD_KEYSTREAM_NXT".NXT_KSTRM_07, X08_OUT_KSTRM => "CHACHA_DWORD_KEYSTREAM_NXT".NXT_KSTRM_08, X09_OUT_KSTRM => "CHACHA_DWORD_KEYSTREAM_NXT".NXT_KSTRM_09, X10_OUT_KSTRM => "CHACHA_DWORD_KEYSTREAM_NXT".NXT_KSTRM_10, X11_OUT_KSTRM => "CHACHA_DWORD_KEYSTREAM_NXT".NXT_KSTRM_11, X12_OUT_KSTRM => "CHACHA_DWORD_KEYSTREAM_NXT".NXT_KSTRM_12, X13_OUT_KSTRM => "CHACHA_DWORD_KEYSTREAM_NXT".NXT_KSTRM_13, X14_OUT_KSTRM => "CHACHA_DWORD_KEYSTREAM_NXT".NXT_KSTRM_14, X15_OUT_KSTRM => "CHACHA_DWORD_KEYSTREAM_NXT".NXT_KSTRM_15)
   END_RUNG
   // the same network as SCL:
   "CHACHA_20_ROUNDS"(X00_IN := "CHACHA_DWORD_DB".X00_CNST0_DWORD,
                      X01_IN := "CHACHA_DWORD_DB".X01_CNST1_DWORD,
                      X02_IN := "CHACHA_DWORD_DB".X02_CNST2_DWORD,
                      X03_IN := "CHACHA_DWORD_DB".X03_CNST3_DWORD,
                      X04_IN := "CHACHA_DWORD_DB".X04_K0_DWORD,
                      X05_IN := "CHACHA_DWORD_DB".X05_K1_DWORD,
                      X06_IN := "CHACHA_DWORD_DB".X06_K2_DWORD,
                      X07_IN := "CHACHA_DWORD_DB".X07_K3_DWORD,
                      X08_IN := "CHACHA_DWORD_DB".X08_K4_DWORD,
                      X09_IN := "CHACHA_DWORD_DB".X09_K5_DWORD,
                      X10_IN := "CHACHA_DWORD_DB".X10_K6_DWORD,
                      X11_IN := "CHACHA_DWORD_DB".X11_K7_DWORD,
                      X12_IN := "CHACHA_DWORD_DB".X12_CNTR0_DWORD,
                      X13_IN := "CHACHA_DWORD_DB".X13_NONCE0_DWORD,
                      X14_IN := "CHACHA_DWORD_DB".X14_NONCE1_DWORD,
                      X15_IN := "CHACHA_DWORD_DB".X15_NONCE2_DWORD,
                      X00_OUT => "CHACHA_DWORD_DB".X00_CNST0_DWORD,
                      X01_OUT => "CHACHA_DWORD_DB".X01_CNST1_DWORD,
                      X02_OUT => "CHACHA_DWORD_DB".X02_CNST2_DWORD,
                      X03_OUT => "CHACHA_DWORD_DB".X03_CNST3_DWORD,
                      X04_OUT => "CHACHA_DWORD_DB".X04_K0_DWORD,
                      X05_OUT => "CHACHA_DWORD_DB".X05_K1_DWORD,
                      X06_OUT => "CHACHA_DWORD_DB".X06_K2_DWORD,
                      X07_OUT => "CHACHA_DWORD_DB".X07_K3_DWORD,
                      X08_OUT => "CHACHA_DWORD_DB".X08_K4_DWORD,
                      X09_OUT => "CHACHA_DWORD_DB".X09_K5_DWORD,
                      X10_OUT => "CHACHA_DWORD_DB".X10_K6_DWORD,
                      X11_OUT => "CHACHA_DWORD_DB".X11_K7_DWORD,
                      X12_OUT => "CHACHA_DWORD_DB".X12_CNTR0_DWORD,
                      X13_OUT => "CHACHA_DWORD_DB".X13_NONCE0_DWORD,
                      X14_OUT => "CHACHA_DWORD_DB".X14_NONCE1_DWORD,
                      X15_OUT => "CHACHA_DWORD_DB".X15_NONCE2_DWORD,
                      X00_OUT_KSTRM => "CHACHA_DWORD_KEYSTREAM".KSTRM_00,
                      X01_OUT_KSTRM => "CHACHA_DWORD_KEYSTREAM".KSTRM_01,
                      X02_OUT_KSTRM => "CHACHA_DWORD_KEYSTREAM".KSTRM_02,
                      X03_OUT_KSTRM => "CHACHA_DWORD_KEYSTREAM".KSTRM_03,
                      X04_OUT_KSTRM => "CHACHA_DWORD_KEYSTREAM".KSTRM_04,
                      X05_OUT_KSTRM => "CHACHA_DWORD_KEYSTREAM".KSTRM_05,
                      X06_OUT_KSTRM => "CHACHA_DWORD_KEYSTREAM".KSTRM_06,
                      X07_OUT_KSTRM => "CHACHA_DWORD_KEYSTREAM".KSTRM_07,
                      X08_OUT_KSTRM => "CHACHA_DWORD_KEYSTREAM".KSTRM_08,
                      X09_OUT_KSTRM => "CHACHA_DWORD_KEYSTREAM".KSTRM_09,
                      X10_OUT_KSTRM => "CHACHA_DWORD_KEYSTREAM".KSTRM_10,
                      X11_OUT_KSTRM => "CHACHA_DWORD_KEYSTREAM".KSTRM_11,
                      X12_OUT_KSTRM => "CHACHA_DWORD_KEYSTREAM".KSTRM_12,
                      X13_OUT_KSTRM => "CHACHA_DWORD_KEYSTREAM".KSTRM_13,
                      X14_OUT_KSTRM => "CHACHA_DWORD_KEYSTREAM".KSTRM_14,
                      X15_OUT_KSTRM => "CHACHA_DWORD_KEYSTREAM".KSTRM_15,
                      ENO => #_w1);
   IF #_w1 THEN
       "CHACHA_20_ROUNDS"(X00_IN := "CHACHA_DWORD_DB".X00_CNST0_DWORD,
                          X01_IN := "CHACHA_DWORD_DB".X01_CNST1_DWORD,
                          X02_IN := "CHACHA_DWORD_DB".X02_CNST2_DWORD,
                          X03_IN := "CHACHA_DWORD_DB".X03_CNST3_DWORD,
                          X04_IN := "CHACHA_DWORD_DB".X04_K0_DWORD,
                          X05_IN := "CHACHA_DWORD_DB".X05_K1_DWORD,
                          X06_IN := "CHACHA_DWORD_DB".X06_K2_DWORD,
                          X07_IN := "CHACHA_DWORD_DB".X07_K3_DWORD,
                          X08_IN := "CHACHA_DWORD_DB".X08_K4_DWORD,
                          X09_IN := "CHACHA_DWORD_DB".X09_K5_DWORD,
                          X10_IN := "CHACHA_DWORD_DB".X10_K6_DWORD,
                          X11_IN := "CHACHA_DWORD_DB".X11_K7_DWORD,
                          X12_IN := "CHACHA_DWORD_DB".X12_CNTR0_DWORD,
                          X13_IN := "CHACHA_DWORD_DB".X13_NONCE0_DWORD,
                          X14_IN := "CHACHA_DWORD_DB".X14_NONCE1_DWORD,
                          X15_IN := "CHACHA_DWORD_DB".X15_NONCE2_DWORD,
                          X00_OUT => "CHACHA_DWORD_DB".X00_CNST0_DWORD,
                          X01_OUT => "CHACHA_DWORD_DB".X01_CNST1_DWORD,
                          X02_OUT => "CHACHA_DWORD_DB".X02_CNST2_DWORD,
                          X03_OUT => "CHACHA_DWORD_DB".X03_CNST3_DWORD,
                          X04_OUT => "CHACHA_DWORD_DB".X04_K0_DWORD,
                          X05_OUT => "CHACHA_DWORD_DB".X05_K1_DWORD,
                          X06_OUT => "CHACHA_DWORD_DB".X06_K2_DWORD,
                          X07_OUT => "CHACHA_DWORD_DB".X07_K3_DWORD,
                          X08_OUT => "CHACHA_DWORD_DB".X08_K4_DWORD,
                          X09_OUT => "CHACHA_DWORD_DB".X09_K5_DWORD,
                          X10_OUT => "CHACHA_DWORD_DB".X10_K6_DWORD,
                          X11_OUT => "CHACHA_DWORD_DB".X11_K7_DWORD,
                          X12_OUT => "CHACHA_DWORD_DB".X12_CNTR0_DWORD,
                          X13_OUT => "CHACHA_DWORD_DB".X13_NONCE0_DWORD,
                          X14_OUT => "CHACHA_DWORD_DB".X14_NONCE1_DWORD,
                          X15_OUT => "CHACHA_DWORD_DB".X15_NONCE2_DWORD,
                          X00_OUT_KSTRM => "CHACHA_DWORD_KEYSTREAM_NXT".NXT_KSTRM_00,
                          X01_OUT_KSTRM => "CHACHA_DWORD_KEYSTREAM_NXT".NXT_KSTRM_01,
                          X02_OUT_KSTRM => "CHACHA_DWORD_KEYSTREAM_NXT".NXT_KSTRM_02,
                          X03_OUT_KSTRM => "CHACHA_DWORD_KEYSTREAM_NXT".NXT_KSTRM_03,
                          X04_OUT_KSTRM => "CHACHA_DWORD_KEYSTREAM_NXT".NXT_KSTRM_04,
                          X05_OUT_KSTRM => "CHACHA_DWORD_KEYSTREAM_NXT".NXT_KSTRM_05,
                          X06_OUT_KSTRM => "CHACHA_DWORD_KEYSTREAM_NXT".NXT_KSTRM_06,
                          X07_OUT_KSTRM => "CHACHA_DWORD_KEYSTREAM_NXT".NXT_KSTRM_07,
                          X08_OUT_KSTRM => "CHACHA_DWORD_KEYSTREAM_NXT".NXT_KSTRM_08,
                          X09_OUT_KSTRM => "CHACHA_DWORD_KEYSTREAM_NXT".NXT_KSTRM_09,
                          X10_OUT_KSTRM => "CHACHA_DWORD_KEYSTREAM_NXT".NXT_KSTRM_10,
                          X11_OUT_KSTRM => "CHACHA_DWORD_KEYSTREAM_NXT".NXT_KSTRM_11,
                          X12_OUT_KSTRM => "CHACHA_DWORD_KEYSTREAM_NXT".NXT_KSTRM_12,
                          X13_OUT_KSTRM => "CHACHA_DWORD_KEYSTREAM_NXT".NXT_KSTRM_13,
                          X14_OUT_KSTRM => "CHACHA_DWORD_KEYSTREAM_NXT".NXT_KSTRM_14,
                          X15_OUT_KSTRM => "CHACHA_DWORD_KEYSTREAM_NXT".NXT_KSTRM_15);
   END_IF;
END_REGION
END_ORGANIZATION_BLOCK